{attribute 'linkalways'} 
{attribute 'no_explicit_call' := 'This FB is a CLASS and must be accessed using methods or properties'}
{attribute 'enable_dynamic_creation'}
FUNCTION_BLOCK IncorrectKeyTypeDeserializationError EXTENDS IncorrectTypeDeserializationError
VAR
	key : T_MAXSTRING;
END_VAR

METHOD FB_init : BOOL
VAR_INPUT
	bInitRetains : BOOL; // if TRUE, the retain variables are initialized (warm start / cold start)
	bInCopyCode : BOOL;  // if TRUE, the instance afterwards gets moved into the copy code (online change)
	DataType : T_MAXSTRING;
	Key : T_MAXSTRING;
END_VAR
THIS^.key := Key;
END_METHOD

PROPERTY PUBLIC Message : T_MAXSTRING
GET
VAR
	messageWithKey : T_MAXSTRING;
END_VAR
messageWithKey := concat(' for key : ',key);
Message := CONCAT(SUPER^.Message, messageWithKey);
END_GET
END_PROPERTY

END_FUNCTION_BLOCK

(* stored: Version 1.1.0.1, ProductVersion 3.1.4024.12
   POU IncorrectKeyTypeDeserializationError: Id {9a3970b9-c7ea-07b0-1329-2628cf8059c8}, SpecialFunc None
   Folder Constructor: Id {20fdd53a-fb6a-0ed0-23dc-1ebce2acc1f1}
   Method FB_init: Id {cdcccc56-d58b-0ae5-1a00-b6039da119de}
   Property Message: Id {60de2e30-c9ce-0f2a-0904-b07880adc046}
   Get Get: Id {43ae9383-042f-0590-15a7-ec14347ef1dc} *)
